(*			
	EVERDE sp. z o.o.
	Rafał Osajda		29.10.2025		TC 4024.66
	Metody do konfiguracji MAchine control wywoływane z MachineConfigure z pomocą przekazanego ITF
*)
INTERFACE ITF_MachineControlConfigure EXTENDS ITF_Base

METHOD AddTopElementFromConfiguration : BOOL
VAR_INPUT
	fbTopElement		: ITF_BaseTopElement;
END_VAR
END_METHOD

END_INTERFACE

(* stored: Version 1.1.0.1
   Itf ITF_MachineControlConfigure: Id {407b3a6e-6e4f-4b87-8313-a53f9cca235d}
   Method AddTopElementFromConfiguration: Id {c458ce8f-1021-07a3-1b12-05adfb9f74f9} *)
